(* IEC 61131-3 sources: mect_apps/TPAC1008/Collaudo_PLC, 8 files *)

(* ---- Collaudo_CAN.gvl ---- *)
(* Global var file *)
VAR_GLOBAL
	ch1_CAN1_IN_DIG_8_1 AT %IB3.4096: BYTE;
	ch1_CAN1_IN_DIG_8_2 AT %IB3.4097: BYTE;
	ch1_CAN1_OUT_DIG_8_1 AT %QB3.4096: BYTE;
	ch1_CAN1_OUT_DIG_8_2 AT %QB3.4097: BYTE;
	ch1_CAN1_IN_AN_1 AT %IW3.8192: INT;
	ch1_CAN1_IN_AN_2 AT %IW3.8194: INT;
	ch1_CAN1_IN_AN_3 AT %IW3.8196: INT;
	ch1_CAN1_IN_AN_4 AT %IW3.8198: INT;
	ch1_CAN1_IN_AN_5 AT %IW3.8200: INT;
	ch1_CAN1_IN_AN_6 AT %IW3.8202: INT;
	ch1_CAN1_IN_AN_7 AT %IW3.8204: INT;
	ch1_CAN1_IN_AN_8 AT %IW3.8206: INT;
	ch1_CAN1_IN_AN_9 AT %IW3.8208: INT;
	ch1_CAN1_IN_AN_10 AT %IW3.8210: INT;
	ch1_CAN1_IN_AN_11 AT %IW3.8212: INT;
	ch1_CAN1_IN_AN_12 AT %IW3.8214: INT;
	ch1_CAN1_IN_AN_13 AT %IW3.8216: INT;
	ch1_CAN1_IN_AN_14 AT %IW3.8218: INT;
	ch1_CAN1_IN_AN_15 AT %IW3.8220: INT;
	ch1_CAN1_IN_AN_16 AT %IW3.8222: INT;
	ch1_CAN1_OUT_AN_1 AT %QW3.8192: INT;
	PLC_CAN1_IN_DIG_8_1 AT %MB0.5380: BYTE;
	PLC_CAN1_IN_DIG_8_2 AT %MB0.5384: BYTE;
	PLC_CAN1_OUT_DIG_8_1 AT %MB0.5388: BYTE;
	PLC_CAN1_OUT_DIG_8_2 AT %MB0.5392: BYTE;
	PLC_CAN1_IN_AN_1 AT %MW0.5396: INT;
	PLC_CAN1_IN_AN_2 AT %MW0.5400: INT;
	PLC_CAN1_IN_AN_3 AT %MW0.5404: INT;
	PLC_CAN1_IN_AN_4 AT %MW0.5408: INT;
	PLC_CAN1_IN_AN_5 AT %MW0.5412: INT;
	PLC_CAN1_IN_AN_6 AT %MW0.5416: INT;
	PLC_CAN1_IN_AN_7 AT %MW0.5420: INT;
	PLC_CAN1_IN_AN_8 AT %MW0.5424: INT;
	PLC_CAN1_IN_AN_9 AT %MW0.5428: INT;
	PLC_CAN1_IN_AN_10 AT %MW0.5432: INT;
	PLC_CAN1_IN_AN_11 AT %MW0.5436: INT;
	PLC_CAN1_IN_AN_12 AT %MW0.5440: INT;
	PLC_CAN1_IN_AN_13 AT %MW0.5444: INT;
	PLC_CAN1_IN_AN_14 AT %MW0.5448: INT;
	PLC_CAN1_IN_AN_15 AT %MW0.5452: INT;
	PLC_CAN1_IN_AN_16 AT %MW0.5456: INT;
	PLC_CAN1_OUT_AN_1 AT %MW0.5460: INT;
END_VAR

(* ---- ImpostazioniCAN1.gvl ---- *)
(* Global var file *)
VAR_GLOBAL
	ch1_CAN1_IN_DIG_8_1 AT %IB3.4096: BYTE;
	ch1_CAN1_IN_DIG_8_2 AT %IB3.4097: BYTE;
	ch1_CAN1_OUT_DIG_8_1 AT %QB3.4096: BYTE;

	ch1_CAN1_OUT_DIG_8_1_7 AT %QX3.4096.7: BOOL;

	ch1_CAN1_OUT_DIG_8_2 AT %QB3.4097: BYTE;
	ch1_CAN1_IN_AN_1 AT %IW3.5396: INT;
	ch1_CAN1_IN_AN_2 AT %IW3.5398: INT;
	ch1_CAN1_IN_AN_3 AT %IW3.5400: INT;
	ch1_CAN1_IN_AN_4 AT %IW3.5402: INT;
	ch1_CAN1_IN_AN_5 AT %IW3.5404: INT;
	ch1_CAN1_IN_AN_6 AT %IW3.5408: INT;
	ch1_CAN1_IN_AN_7 AT %IW3.5410: INT;
	ch1_CAN1_IN_AN_8 AT %IW3.5412: INT;
	ch1_CAN1_IN_AN_9 AT %IW3.5414: INT;
	ch1_CAN1_IN_AN_10 AT %IW3.5416: INT;
	ch1_CAN1_IN_AN_11 AT %IW3.5418: INT;
	ch1_CAN1_IN_AN_12 AT %IW3.5420: INT;
	ch1_CAN1_IN_AN_13 AT %IW3.5422: INT;
	ch1_CAN1_IN_AN_14 AT %IW3.5424: INT;
	ch1_CAN1_IN_AN_15 AT %IW3.5426: INT;
	ch1_CAN1_IN_AN_16 AT %IW3.5428: INT;
	ch1_CAN1_OUT_AN_1 AT %QW3.8192: INT;
	PLC_CAN1_IN_DIG_8_1 AT %MB0.21200: BYTE;

	PLC_CAN1_IN_DIG_8_2 AT %MB0.21204: BYTE;
	PLC_CAN1_OUT_DIG_8_1 AT %MB0.21208: BYTE;
	PLC_CAN1_OUT_DIG_8_1_0 AT %MX0.21208.0: BOOL;
	PLC_CAN1_OUT_DIG_8_1_1 AT %MX0.21208.1: BOOL;
	PLC_CAN1_OUT_DIG_8_1_2 AT %MX0.21208.2: BOOL;
	PLC_CAN1_OUT_DIG_8_1_3 AT %MX0.21208.3: BOOL;
	PLC_CAN1_OUT_DIG_8_1_4 AT %MX0.21208.4: BOOL;
	PLC_CAN1_OUT_DIG_8_1_5 AT %MX0.21208.5: BOOL;
	PLC_CAN1_OUT_DIG_8_1_6 AT %MX0.21208.6: BOOL;
	PLC_CAN1_OUT_DIG_8_1_7 AT %MX0.21208.7: BOOL;

	PLC_CAN1_OUT_DIG_8_2 AT %MB0.21212: BYTE;

	PLC_CAN1_IN_AN_1 AT %MW0.21216: INT;
	PLC_CAN1_IN_AN_2 AT %MW0.21220: INT;
	PLC_CAN1_IN_AN_3 AT %MW0.21224: INT;
	PLC_CAN1_IN_AN_4 AT %MW0.21228: INT;
	PLC_CAN1_IN_AN_5 AT %MW0.21232: INT;
	PLC_CAN1_IN_AN_6 AT %MW0.21236: INT;
	PLC_CAN1_IN_AN_7 AT %MW0.21240: INT;
	PLC_CAN1_IN_AN_8 AT %MW0.21244: INT;
	PLC_CAN1_IN_AN_9 AT %MW0.21248: INT;
	PLC_CAN1_IN_AN_10 AT %MW0.21252: INT;
	PLC_CAN1_IN_AN_11 AT %MW0.21256: INT;
	PLC_CAN1_IN_AN_12 AT %MW0.21260: INT;
	PLC_CAN1_IN_AN_13 AT %MW0.21264: INT;
	PLC_CAN1_IN_AN_14 AT %MW0.21268: INT;
	PLC_CAN1_IN_AN_15 AT %MW0.21272: INT;
	PLC_CAN1_IN_AN_16 AT %MW0.21276: INT;
	PLC_CAN1_OUT_AN_1 AT %MW0.21280: INT;
END_VAR

(* ---- fb_HW119_Init.st ---- *)
(*[[
]]*)
FUNCTION_BLOCK fb_HW119_Init
#import "Resource1.gvl"
#import "crosstable.gvl"
VAR_INPUT
	TIPO:UINT;
END_VAR
VAR
	k:WORD;
	i:DINT;
END_VAR
IF TIPO = 0 	THEN
	FOR i:=0 TO DimCrossTable-1	DO

		TRIGGER01 := 0;
		CrossTable[i].Enable:=0;
		CrossTable[i].Plc:=FALSE;
		CrossTable[i].Tag:='';
		CrossTable[i].Types:=0;
		CrossTable[i].Decimal:=0;
		CrossTable[i].Protocol:=0;
		CrossTable[i].IPAddress:='';
		CrossTable[i].Port:=0;
		CrossTable[i].NodeId:=0;
		CrossTable[i].Address:=0;
		CrossTable[i].Block:=0;
		CrossTable[i].NReg:=0;
		CrossTable[i].Handle:=0;
		CrossTable[i].OldVal:=0;
		CrossTable[i].Error:=1;
		K:=ARRAY_QUEUE[i+1];
		ARRAY_QUEUE_OUTPUT[i+1]:=0;
		ARRAY_STATES[i+1]:=0;

	END_FOR;
	CrossTableState:=TRUE;
	CommEnabled:=FALSE;
	RTUProtocol_ON:=FALSE;
	TCPProtocol_ON:=FALSE;
	TCPRTUProtocol_ON:=FALSE;

ELSIF  TIPO = 1 	THEN
	FOR i:=0 TO 159	DO

		ALCrossTable[i].ALType:=FALSE;
		ALCrossTable[i].ALTag:='';
		ALCrossTable[i].ALSource:='';
		ALCrossTable[i].ALCompareVar:='';
		ALCrossTable[i].ALCompareVal:=0;
		ALCrossTable[i].ALOperator:=0;
		ALCrossTable[i].ALFilterTime:=0;
	END_FOR;
	ALCrossTableState:=TRUE;
 END_IF;
END_FUNCTION_BLOCK

(* ---- fb_HW119_PLCreadVar.st ---- *)
(*[[
]]*)
FUNCTION_BLOCK fb_HW119_PLCreadVar
#import "Resource1.gvl"
#import "crosstable.gvl"
VAR_INPUT
	ReadVar:STRING;			(*	Mnemonico della variabile da leggere	*)
END_VAR
VAR_OUTPUT
	ERR:BOOL;				(*	Segnala errore nell'esecuzione del blocco funzione	*)
	VarValue:DWORD;			(*	Valore letto	*)
END_VAR
VAR
	ReadingAddr:WORD;

END_VAR
(*
		Blocco funzione per la lettura di una variabile attraverso il PLC di controllo

*)

	ReadingAddr:=HW119_GetAddr(ReadVar);
	IF ReadingAddr =16#FFFF THEN
		ERR:=TRUE;
		HW119_ERR[4]:=3;
	ELSE
		VarValue:=ARRAY_CROSSTABLE_INPUT[WORD_TO_INT(ReadingAddr)];
		ARRAY_STATES[WORD_TO_INT(ReadingAddr)]=0;
		HW119_ERR[4]:=2;
	END_IF;
END_FUNCTION_BLOCK

(* ---- fb_HW119_PLCsync.st ---- *)
(*[[
]]*)
FUNCTION_BLOCK fb_HW119_PLCsync
#import "Resource1.gvl"
#import "crosstable.gvl"
VAR_INPUT
END_VAR
VAR
	IndexPLC:UINT;
	I:INT;
	RW:WORD;
	addr:INT;
	duster:UINT:=1;
END_VAR

		IF duster < DINT_TO_UINT(DimCrossTable) AND duster < maxQueue THEN
			RW:=ARRAY_QUEUE[duster] AND QueueRWMask;
			IF  RW  = 0 AND  ARRAY_QUEUE_OUTPUT[duster]=STATO_BUSY_WRITE  THEN
				ARRAY_QUEUE_OUTPUT[duster]:=0;
			END_IF;
			duster:=duster+1;
		ELSE
			duster:=1;
		END_IF;
		(* Rileva la prima variabile da leggere della cross table*)
		IF IndexPLC < DINT_TO_UINT(DimCrossTable) THEN
			IndexPLC:=IndexPLC+1;
			RW:=ARRAY_QUEUE[IndexPLC] AND QueueRWMask;
			addr:=WORD_TO_INT(ARRAY_QUEUE[IndexPLC] AND QueueAddressMask);
			IF addr < DINT_TO_INT(DimCrossTable)	THEN
				IF  RW  = 0 AND  ARRAY_QUEUE_OUTPUT[IndexPLC]=STATO_BUSY_WRITE AND CrossTable[addr].Protocol = 100 THEN
					ARRAY_QUEUE_OUTPUT[IndexPLC]:=0;
				ELSIF RW =0 AND addr =0 THEN
					ARRAY_QUEUE_OUTPUT[IndexPLC]:=0;
					IndexPLC:=0;
				ELSIF ( RW  = WRITE OR  RW  = WRITE_RIC_SINGLE OR RW=WRITE_MULTIPLE) AND  ARRAY_QUEUE_OUTPUT[IndexPLC]<>STATO_BUSY_WRITE AND CrossTable[addr].Protocol = 100 THEN
					ARRAY_QUEUE_OUTPUT[IndexPLC]:=STATO_BUSY_WRITE;
					IF (RW  = WRITE) OR (RW  = WRITE_RIC_SINGLE) THEN
						ARRAY_CROSSTABLE_INPUT[addr]:=ARRAY_CROSSTABLE_OUTPUT[addr];
					ELSE
						FOR I:=0 TO CrossTable[addr].NReg - 1 DO			(*	copia dei valori da leggere nel buffer di comunicazione	*)
							ARRAY_CROSSTABLE_INPUT[addr+I]:=ARRAY_CROSSTABLE_OUTPUT[addr+I];
							CrossTable[addr+I].Error:=0;							(*indica che la variabile è aggiornata*)
						END_FOR;
					END_IF;
				END_IF;
			END_IF;
		ELSE
			IndexPLC:=0;
		END_IF;

END_FUNCTION_BLOCK

(* ---- fb_TPAC_tic.st ---- *)
(*[[
]]*)
FUNCTION_BLOCK fb_TPAC_tic
	#import "TPACLocaIO.gvl"
VAR_INPUT
	tic:TIME;
END_VAR
VAR
END_VAR
	PLC_time:=PLC_time + 0.001 * TIME_TO_REAL(tic);
	IF PLC_time > 86400.0 THEN
		PLC_time:=0.0;
	END_IF;
	if PLC_time > 10.0 then
		PLC_timeMax := PLC_time;
		PLC_timeMin := PLC_time - 10.0;
	else
		PLC_timeMax := 10.0;
		PLC_timeMin := 0.0;
	end_if;
END_FUNCTION_BLOCK

(* ---- PLC.st ---- *)
(*[[
]]*)
PROGRAM PLC
#import "Resource1.gvl"
#import "crosstable.gvl"
#import "TPACLocaIO.gvl" (* <---= *)
#import "Collaudo_CAN.gvl"
#import "LIO_TPAC1006.gvl"
VAR
	fb_HW119_PLCwriteVar_Inst : fb_HW119_PLCwriteVar;
	values : ARRAY [0..15] OF DWORD;
	TIMER1:TON;
	TIMER2:TON;
END_VAR;
values[0]:=1;
fb_HW119_PLCwriteVar_Inst(VARIABLE := 'Modbus_1', VALUES := values, Nregs := 1);
IF FALSE THEN
	ch1_CAN1_OUT_DIG_8_1:=0;
END_IF;
TIMER1(in:=TRUE,PT:=T#1s);
IF TIMER1.Q THEN
	TIMER1(in:=FALSE,PT:=T#1s);
	IF ch1_CAN1_OUT_DIG_8_1 = 16#01 THEN
		ch1_CAN1_OUT_DIG_8_1:=16#01;
	ELSE
		ch1_CAN1_OUT_DIG_8_1:=16#00;
	END_IF;
end_if;
PLC_CAN1_IN_AN_1:=ch1_CAN1_IN_AN_1;
PLC_CAN1_IN_AN_2:=ch1_CAN1_IN_AN_2;
PLC_CAN1_IN_AN_3:=ch1_CAN1_IN_AN_3;
PLC_CAN1_IN_AN_4:=ch1_CAN1_IN_AN_4;
PLC_CAN1_IN_AN_5:=ch1_CAN1_IN_AN_5;
PLC_CAN1_IN_AN_6:=ch1_CAN1_IN_AN_6;
PLC_CAN1_IN_AN_7:=ch1_CAN1_IN_AN_7;
PLC_CAN1_IN_AN_8:=ch1_CAN1_IN_AN_8;
PLC_CAN1_IN_AN_9:=ch1_CAN1_IN_AN_9;
PLC_CAN1_IN_AN_10:=ch1_CAN1_IN_AN_10;
PLC_CAN1_IN_AN_11:=ch1_CAN1_IN_AN_11;
PLC_CAN1_IN_AN_12:=ch1_CAN1_IN_AN_12;
PLC_CAN1_IN_AN_13:=ch1_CAN1_IN_AN_13;
PLC_CAN1_IN_AN_14:=ch1_CAN1_IN_AN_14;
PLC_CAN1_IN_AN_15:=ch1_CAN1_IN_AN_15;
PLC_CAN1_IN_AN_16:=ch1_CAN1_IN_AN_16;

END_PROGRAM

(* ---- RTU_Communication.st ---- *)
(*[[
]]*)
PROGRAM RTU_Communication
#import "Resource1.gvl"
#import "crosstable.gvl"
VAR
	HeadAddr:INT;
	ReadWrite:WORD;
	IndexProt_i:ARRAY [0..4] OF INT;
	TON_0:TON;
	TON_1:TON;
	TON_2:TON;
	TON_3:TON;
	BusAccess:fb_HW119_MODBUS;
	FirstCy:BOOL;
	dummy:WORD;
	Enablei: ARRAY [0..3] OF BOOL;
	pointer:INT;
	FlagPrimoCiclo:BOOL;
	Retry:BOOL:=FALSE;
	Protocollo:UINT:=RTU;
	timeCount:ARRAY [0..4] OF UDINT;
	zeroCount:ARRAY [0..4] OF UDINT;
	deltaT: ARRAY [0..4] OF DINT;
	RicettaON:BOOL;
	LastID:INT;
	FirstID:INT;
	I:INT;
	Start:ARRAY [0..4] OF BOOL;
	k:dword;
	j:dword;
	plcCylce:UDINT:=10;
	TIC:UDINT:=0;
	TAC:UDINT:=0;
	tailPoint:INT;
END_VAR
IF NOT FirstCy THEN
	dummy:=	WD_Disable('Task2_RTU');
	timeCount[0]:=0;
	timeCount[1]:=0;
	timeCount[2]:=0;
	deltaT[0]:=0;
	deltaT[1]:=0;
	deltaT[2]:=0;
	FirstCy:=TRUE;
END_IF;
TAC:=TAC+1;
TON_0(IN := TRUE,PT := INT_TO_TIME(CommParameters[Protocollo+1].Tmin));
(*				TON_1(IN := TRUE,PT := DINT_TO_TIME(Talta+deltaT[0]));
				TON_2(IN := TRUE,PT := DINT_TO_TIME(Tmedia+deltaT[1]));
				TON_3(IN := TRUE,PT := DINT_TO_TIME(Tbassa+deltaT[2]));
*)
				TON_1(IN := TRUE,PT := DINT_TO_TIME(Talta));
				TON_2(IN := TRUE,PT := DINT_TO_TIME(Tmedia));
				TON_3(IN := TRUE,PT := DINT_TO_TIME(Tbassa));

IF 	TON_0.Q THEN																(* controlla se TIMER Tmin scaduto	*)
	TRIGGER02:=1;
	TRIGGER01:=1;
	TIC:=TIC+1;
	TON_0(In:=FALSE);

	IF Reset_RTU =1 THEN
		FOR I:=1 TO 64 DO
			CounterRTU[I]:=0;
		 END_FOR;
		RTUBlackList_ERROR_WORD:=0;
		RTUComm_ERROR_WORD:=0;
		BlackListRTUL:=0;
		BlackListRTUH:=0;
		CommErrRTUL:=0;
		CommErrRTUH:=0;
		ERROR_FLAG:=ERROR_FLAG AND 16#FFFE;
	END_IF;
	IF NOT Retry THEN
		IF RTURequestPLCWrite > 0 (*AND
			(MOD(TIC ,3)=0  OR (mod(tic,3)=1 and RichiestaScrittura=0))*) THEN											(* controlla seci sono richieste di scrittura da parte del PLC	*)

			pointer:=4;
			FlagPrimoCiclo:=FALSE;
			IndexProt_i[pointer]:=0;
			HeadAddr:=WORD_TO_INT(LocalRTUQueue[IndexRTUQueueGet]);		(*inizializza i parametri da assegnare al blocco funzione*)
			IF CrossTable[HeadAddr].Counter=1 THEN
				ReadWrite:=WRITE_SINGLE;											(*inizializza i parametri da assegnare al blocco funzione*)
			ELSE
				ReadWrite:=WRITE_MULTIPLE;											(*inizializza i parametri da assegnare al blocco funzione*)
			END_IF;

			RTURequestPLCWrite:=RTURequestPLCWrite-1;							(* incrementa il contatore delle scritture effettuate*)
			IndexRTUQueueGet:=IndexRTUQueueGet+1;								(* incrementa il puntatore alla coda *)
			IF IndexRTUQueueGet > MaxLocalQueue THEN
				IndexRTUQueueGet:=0;
			END_IF;
		ELSE
			IF  (RichiestaScrittura=1 (*AND MOD(TIC ,7)< 6*)) THEN										(* controlla se ci sono richieste di SCRITTURA da parte HMI*)

				IF FlagPrimoCiclo = FALSE THEN									(* controlla se è il primo ingrsso nel ramo a seguito dell'interrupt*)
					FlagPrimoCiclo:=TRUE;										(* Prima richiesta di scrittura => azzero l'indice della coda 	*)
					IndexProt_i[3]:=0;											(* per eseguire le scritture nella sequenza di arrivo		  	*)
					pointer:=3;
				END_IF;
				REPEAT 															(* Rileva la succssiva variabile a cui accedere nella coda			*)
					IF IndexProt_i[3] < DINT_TO_INT(DimCrossTable) THEN
						IndexProt_i[3]:=IndexProt_i[3]+1;
						ReadWrite:=ARRAY_QUEUE[IndexProt_i[3]] AND QueueRWMask;
						HeadAddr:=WORD_TO_INT(ARRAY_QUEUE[IndexProt_i[3]] AND QueueAddressMask);
						IF HeadAddr < DINT_TO_INT(DimCrossTable) 	THEN
							IF  (ReadWrite = 0  ) OR ( (CrossTable[HeadAddr].Protocol = Protocollo) AND ReadWrite>=WRITE AND (ARRAY_QUEUE_OUTPUT[IndexProt_i[3]]<>STATO_BUSY_WRITE) )   THEN

								IF ReadWrite = 0 THEN
									ARRAY_QUEUE_OUTPUT[IndexProt_i[3]]:=0;
									IF HeadAddr = 0 THEN
										IndexProt_i[3]:=0;
									END_IF;

								ELSIF ReadWrite = WRITE_RIC_SINGLE  OR ReadWrite = WRITE_RIC_MULTIPLE  THEN
									IF NOT RicettaON THEN
										FirstID:=IndexProt_i[3];
										RicettaON:=TRUE;
									END_IF;

									LastID:=IndexProt_i[3];
								END_IF;
								IF ReadWrite>=WRITE THEN
									timeCount[4]:=TIC -zeroCount[4];
									zeroCount[4]:=TIC;
									tailPoint:=IndexProt_i[3];
								END_IF;

								EXIT;
							ELSIF ReadWrite = 0 and HeadAddr>0 THEN
								ARRAY_QUEUE_OUTPUT[IndexProt_i[3]]:=0;
							END_IF;
						END_IF;
					ELSE
						IndexProt_i[3]:=0;
					END_IF;
				UNTIL  FALSE
				END_REPEAT;
			ELSIF RicettaON AND RichiestaScrittura=0 THEN
				RicettaON:=FALSE;
				FlagPrimoCiclo:=FALSE;
				FOR I:=1 TO  LastID DO
 					ARRAY_QUEUE_OUTPUT[I]:=0;
				END_FOR;
			ELSE																			(* richieste di LETTURE	*)
				IF  RichiestaScrittura=0	THEN
					FlagPrimoCiclo:=FALSE;										(* azzera l'akwnoledge dell'interrupt*)
					IF tailPoint> 0 THEN
						FOR I:=tailPoint TO 0 by -1 do
							ARRAY_QUEUE_OUTPUT[tailPoint]:=0;
							IF (ARRAY_QUEUE[tailPoint] AND QueueRWMask) > 0 THEN
								EXIT;
							END_IF;
						END_FOR;
					 	tailPoint:=0;
					END_IF;

				END_IF;
			END_IF;
			IF  RichiestaScrittura=0 (*or   (RichiestaScrittura=1 and ReadWrite=0) *) then
				IF TON_1.Q OR Enablei[0]=TRUE THEN							(* scaduto il timer ad alta priorità esegue le letture *)
					IF Enablei[0]=FALSE THEN
						TON_1(IN := FALSE);									(* riarma il timer*)
						Start[0]:=TRUE;
						zeroCount[0]:=TAC;
						deltaT[0]:=UDINT_TO_DINT(timeCount[0]*plcCylce)-Talta;
						IF deltaT[0] <= 0 THEN
							deltaT[0]:=0;
						ELSE
							deltaT[0]:=REAL_TO_DINT(DINT_TO_REAL(deltaT[0])*1.2);
						END_IF;
					END_IF;
					pointer:=0;
					Enablei[0]:=TRUE;
				ELSIF TON_2.Q OR Enablei[1]=TRUE THEN						(* scaduto il timer ad media priorità esegue le letture *)
					IF Enablei[1]=FALSE THEN
						TON_2(IN := FALSE);									(* riarma il timer*)
						Start[1]:=TRUE;
						zeroCount[1]:=TAC;
						deltaT[1]:=UDINT_TO_DINT(timeCount[1]*plcCylce)-Tmedia;
						IF deltaT[1] < 0 THEN
							deltaT[1]:=0;
						ELSE
							deltaT[1]:=REAL_TO_DINT(DINT_TO_REAL(deltaT[1])*1.2);
						END_IF;
					END_IF;
					TON_2(IN := FALSE);										(* riarma il timer*)
					pointer:=1;
					Enablei[1]:=TRUE;
				ELSIF TON_3.Q OR Enablei[2]=TRUE THEN						(* scaduto il timer ad media priorità esegue le letture *)
					IF Enablei[2]=FALSE THEN
						TON_3(IN := FALSE);										(* riarma il timer*)
						Start[2]:=TRUE;
						zeroCount[2]:=TAC;
						deltaT[2]:=UDINT_TO_DINT(timeCount[2]*plcCylce)-Tbassa;
						IF deltaT[2] < 0 THEN
							deltaT[2]:=0;
						ELSE
							deltaT[2]:=REAL_TO_DINT(DINT_TO_REAL(deltaT[2])*1.2);
						END_IF;
					END_IF;
					pointer:=2;
					Enablei[2]:=TRUE;
				END_IF;
				IF Enablei[0] OR Enablei[1] OR Enablei[2] THEN
					REPEAT 															(* Rileva la prima variabile da leggere della cross table*)
						IF IndexProt_i[pointer] < DINT_TO_INT(DimCrossTable) THEN
							IndexProt_i[pointer]:=IndexProt_i[pointer]+1;
							ReadWrite:=ARRAY_QUEUE[IndexProt_i[pointer]] AND QueueRWMask;
							HeadAddr:=WORD_TO_INT(ARRAY_QUEUE[IndexProt_i[pointer]] AND QueueAddressMask);
							IF HeadAddr < DINT_TO_INT(DimCrossTable) 	THEN
								IF ((ReadWrite = 0) OR (CrossTable[HeadAddr].Protocol = Protocollo) AND (CrossTable[HeadAddr].Enable = pointer+1) )    THEN
									IF ReadWrite = 0 THEN
										Enablei[pointer]:=FALSE;
										timeCount[pointer]:=TAC-zeroCount[pointer];
										ARRAY_QUEUE_OUTPUT[IndexProt_i[pointer]]:=0;
										IF HeadAddr = 0 THEN
											IndexProt_i[pointer]:=0;
										END_IF;
									END_IF;
									EXIT;
								END_IF;
							END_IF;
						ELSE
							IndexProt_i[pointer]:=0;
						END_IF;
					UNTIL  FALSE
					END_REPEAT;
				ELSE
					ReadWrite:=0;
				END_IF;

			END_IF;
		END_IF;
	END_IF;
	IF ReadWrite > 0 THEN
		IF Crosstable[HeadAddr].NodeId > 0 AND Crosstable[HeadAddr].NodeId < 64 THEN

			IF RTUListDevices[BYTE_TO_INT(Crosstable[HeadAddr].NodeId)].BlackListed < 2  THEN			(* controlla se il device non è in blacklist*)
				BusAccess(Protocol:='RTU',Index:=IndexProt_i[pointer],address:=HeadAddr,RdWr:=ReadWrite);		(* effettua l'accesso al bus*)
				TON_0(IN := TRUE,PT := INT_TO_TIME(CommParameters[Protocollo+1].Tmin));						(* riarmo di Tmin*)
				IF BusAccess.Error > 0  THEN																(* controlla sec'è stato un errore di comuicazione*)
					ERROR_FLAG:=ERROR_FLAG OR 16#1;
					CounterRTU[BYTE_TO_INT(Crosstable[HeadAddr].NodeId)]:=UDINT_TO_WORD(WORD_TO_UDINT(CounterRTU[BYTE_TO_INT(Crosstable[HeadAddr].NodeId)])+1);
					IF BusAccess.Error = CommError THEN
						RTUComm_ERROR_WORD:=1;
						IF BYTE_TO_INT(Crosstable[HeadAddr].NodeId) > 32 THEN
							CommErrRTUH:=CommErrRTUH OR SHL(16#1,BYTE_TO_INT(Crosstable[HeadAddr].NodeId) -33);
						ELSE
							CommErrRTUL:=CommErrRTUL OR SHL(16#1,BYTE_TO_INT(Crosstable[HeadAddr].NodeId)-1 );
						END_IF;
						Retry:=FALSE;
					ELSIF BusAccess.Error = TimeoutError  THEN		(* controlla se c'è stato un erore di timeout*)
						Retry:=TRUE;							(* imposta il flag retry a TRUE in modo da effettuare le ripetizioni *)
						RTUListDevices[BYTE_TO_INT(Crosstable[HeadAddr].NodeId)].RetryCounter:=RTUListDevices[BYTE_TO_INT(Crosstable[HeadAddr].NodeId)].RetryCounter+1;
						IF RTUListDevices[BYTE_TO_INT(Crosstable[HeadAddr].NodeId)].RetryCounter >= NumberOfFails THEN
							RTUListDevices[BYTE_TO_INT(Crosstable[HeadAddr].NodeId)].BlackListed:=RTUListDevices[BYTE_TO_INT(Crosstable[HeadAddr].NodeId)].BlackListed+1;
							RTUListDevices[BYTE_TO_INT(Crosstable[HeadAddr].NodeId)].JumpRead:=BYTE_TO_INT(FailDivisor);
							Retry:=FALSE;
							IF RTUListDevices[BYTE_TO_INT(Crosstable[HeadAddr].NodeId)].BlackListed > 1 THEN
								RTUBlackList_ERROR_WORD:=1;

								IF BYTE_TO_INT(Crosstable[HeadAddr].NodeId) > 32 THEN
									BlackListRTUH:=BlackListRTUH OR SHL(16#1,BYTE_TO_INT(Crosstable[HeadAddr].NodeId) -33);
								ELSE
									k:=SHL(16#1,BYTE_TO_INT(Crosstable[HeadAddr].NodeId)-1 );
									BlackListRTUL:=BlackListRTUL OR k;
								END_IF;
							END_IF;
						END_IF;
					END_IF;
				ELSE

					Retry:=FALSE;
					IF BYTE_TO_INT(Crosstable[HeadAddr].NodeId) > 32 THEN
						CommErrRTUH:=CommErrRTUH AND ROL(16#FFFFFFFE,BYTE_TO_INT(Crosstable[HeadAddr].NodeId) -33);
						BlackListRTUH:=BlackListRTUH AND ROL(16#FFFFFFFE,BYTE_TO_INT(Crosstable[HeadAddr].NodeId) -33);
					ELSE
						CommErrRTUL:=CommErrRTUL AND ROL(16#FFFFFFFE,BYTE_TO_INT(Crosstable[HeadAddr].NodeId)-1 );
						k:=ROL(16#FFFFFFFE,BYTE_TO_INT(Crosstable[HeadAddr].NodeId)-1 );
						j:=BlackListRTUL;
						j:=j AND k;
						BlackListRTUL:=j;
					END_IF;
					IF CommErrRTUH =0 AND CommErrRTUl = 0 THEN
						RTUComm_ERROR_WORD:=0;
					END_IF;
					IF BlackListRTUH =0 AND BlackListRTUL = 0 THEN
						RTUBlackList_ERROR_WORD:=0;
					END_IF;

					RTUListDevices[BYTE_TO_INT(Crosstable[HeadAddr].NodeId)].BlackListed:=0;
					RTUListDevices[BYTE_TO_INT(Crosstable[HeadAddr].NodeId)].RetryCounter:=0;
				END_IF;
			ELSE
				RTUListDevices[BYTE_TO_INT(Crosstable[HeadAddr].NodeId)].JumpRead:=RTUListDevices[BYTE_TO_INT(Crosstable[HeadAddr].NodeId)].JumpRead-1;
				IF RTUListDevices[BYTE_TO_INT(Crosstable[HeadAddr].NodeId)].JumpRead <= 0 THEN
					RTUListDevices[BYTE_TO_INT(Crosstable[HeadAddr].NodeId)].BlackListed:=1;
					Retry:=TRUE;
				END_IF;
			END_IF;
		END_IF;
	END_IF;
END_IF;
END_PROGRAM
